// TIA Portal V20 export
DATA_BLOCK "DB_Config"   // DB3
TITLE = DB_Config
{ S7_Optimized_Access := 'TRUE' }
AUTHOR : Gemini
// stored: MemoryReserve 100
   VAR
      MaxMotors : Int;
      CycleTime : Real;
      PlantName : String;
   END_VAR
BEGIN
END_DATA_BLOCK
